PROGRAM p_ModbusRx_OutputCoils
VAR
	
END_VAR

HOMS1_XGantry.PAxis.bTwkFwd:=mb_Output_Coils[50];
HOMS1_XGantry.PAxis.bTwkBwd:=mb_Output_Coils[51];
HOMS1_XGantry.SAxis.bTwkFwd:=mb_Output_Coils[52];
HOMS1_XGantry.SAxis.bTwkBwd:=mb_Output_Coils[53];
HOMS1_YGantry.PAxis.bTwkFwd:=mb_Output_Coils[54];
HOMS1_YGantry.PAxis.bTwkBwd:=mb_Output_Coils[55];
HOMS1_YGantry.SAxis.bTwkFwd:=mb_Output_Coils[56];
HOMS1_YGantry.SAxis.bTwkBwd:=mb_Output_Coils[57];
HOMS1_Pitch.Axis.bTwkFwd:=mb_Output_Coils[58];
HOMS1_Pitch.Axis.bTwkBwd:=mb_Output_Coils[59];
HOMS2_XGantry.PAxis.bTwkFwd:=mb_Output_Coils[60];
HOMS2_XGantry.PAxis.bTwkBwd:=mb_Output_Coils[61];
HOMS2_XGantry.SAxis.bTwkFwd:=mb_Output_Coils[62];
HOMS2_XGantry.SAxis.bTwkBwd:=mb_Output_Coils[63];
HOMS2_YGantry.PAxis.bTwkFwd:=mb_Output_Coils[64];
HOMS2_YGantry.PAxis.bTwkBwd:=mb_Output_Coils[65];
HOMS2_YGantry.SAxis.bTwkFwd:=mb_Output_Coils[66];
HOMS2_YGantry.SAxis.bTwkBwd:=mb_Output_Coils[67];
HOMS2_Pitch.Axis.bTwkFwd:=mb_Output_Coils[68];
HOMS2_Pitch.Axis.bTwkBwd:=mb_Output_Coils[69];
HOMS1_Pitch.Piezo.xEnable:=mb_Output_Coils[70];
HOMS1_Pitch.Piezo.xStop:=mb_Output_Coils[71];
HOMS2_Pitch.Piezo.xEnable:=mb_Output_Coils[72];
HOMS2_Pitch.Piezo.xStop:=mb_Output_Coils[73];
HOMS1_XGantry.xUncouple:=mb_Output_Coils[74];
HOMS1_YGantry.xUncouple:=mb_Output_Coils[75];
HOMS2_XGantry.xUncouple:=mb_Output_Coils[76];
HOMS2_YGantry.xUncouple:=mb_Output_Coils[77];
HOMS1_Bender.bTwkFwd:=mb_Output_Coils[78];
HOMS1_Bender.bTwkBwd:=mb_Output_Coils[79];

END_PROGRAM

(* stored: Version 1.1.0.1, ProductVersion 3.1.4020.12
   POU p_ModbusRx_OutputCoils: Id {943c36cb-adb4-42b1-982e-b281da4eed9b}, SpecialFunc None *)
